VAR_GLOBAL
    (*
      PLC-side ring buffer logger to avoid ADS per-sample reads.

      Design:
        - MAIN (2ms task) writes a fixed-size record into a byte ring buffer.
        - PC reads Head and Buffer bytes via ADS and reconstructs records.
        - If PC is too slow and overrun happens, OverrunCount increments.

      Record layout (little-endian):
        u32 magic = 0x56424D31 ('VBM1')
        u32 seq
        u32 t_us (monotonic from cycle count * 2000us)
        i16 pressure_raw
        i16 torque_raw
        i32 pd33_abs_raw
        i32 pd33_rel_raw
        i16 vib_acc_x_raw
        i16 vib_acc_y_raw
        i16 vib_acc_z_raw
        i16 vib_vel_x_raw
        i16 vib_vel_y_raw
        i16 vib_vel_z_raw
        i16 vib_temp_raw
        i16 vib_disp_x_raw
        i16 vib_disp_y_raw
        i16 vib_disp_z_raw
        i16 vib_freq_x_raw
        i16 vib_freq_y_raw
        i16 vib_freq_z_raw
        u8  valves (bit0..3)
        u8  flags (bit0=pd33_comm_ok, bit1=vibration_comm_ok)
        u16 reserved
      Total: 54 bytes per record
    *)

    Enable : BOOL := FALSE;
    Reset : BOOL := FALSE;

    // Ring buffer state (byte indices)
    Head : UDINT; // next write index (monotonic, wraps by modulo on read side)
    Tail : UDINT; // PC should update this as "consumed" index to prevent Overrun

    OverrunCount : UDINT;
    DropCount : UDINT;

    Seq : UDINT;

    // Constants
    RecordSize : UDINT := 54;
    BufferSize : UDINT := 54 * 4096; // 221,184 bytes (~8.2s at 500Hz)

    Buffer : ARRAY [0..(54*4096)-1] OF USINT;
END_VAR

(* stored: Version 1.1.0.1, ProductVersion 3.1.4024.13
   GVL GVL_DataLogger: Id {33d4d6de-2c48-4d5b-bc5d-d0e2d4a3b45b} *)
